SUBAPPLICATION Uebung_039b (* Spiegelabfolge V2 mit Schrittkette *)
  (* Standard: 61499-2; Description: Copyright (c) 2023 Meisterschulen am Ostbahnhof This program and the accompanying materials are made available under the terms of the Eclipse Public License 2.0 which is available at https://www.eclipse.org/legal/epl-2.0/ SPDX-License-Identifier: EPL-2.0 *)
  (* Version 1.0, 2023-10-23, Franz Höpfinger, Meisterschulen am Ostbahnhof, initial API and implementation and/or initial documentation *)
  PACKAGE Uebungen;
  IMPORT Uebungen::const::UT::DefaultPool::SoftKey_F1;
  IMPORT logiBUS::io::DQ::logiBUS_DO::Output_Q1;
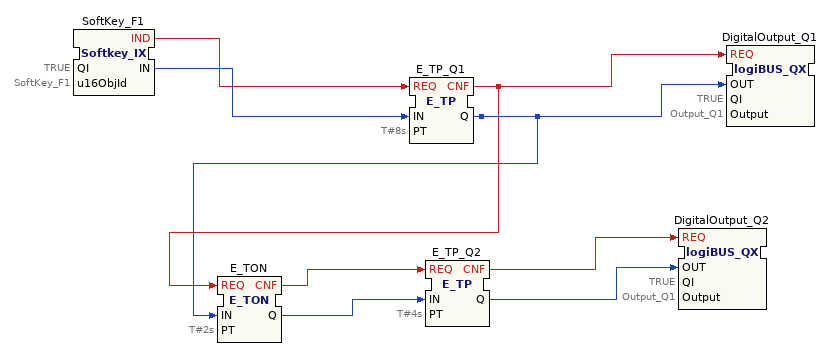
  FBS
    DigitalOutput_Q1 : logiBUS::io::DQ::logiBUS_QX(QI := TRUE, Output := Output_Q1);
    DigitalOutput_Q2 : logiBUS::io::DQ::logiBUS_QX(QI := TRUE, Output := Output_Q1);
    SoftKey_F1 : isobus::UT::io::Softkey::Softkey_IX(QI := TRUE, u16ObjId := SoftKey_F1);
    E_TP_Q1 : iec61499::events::timers::E_TP(PT := T#8s);
    E_TP_Q2 : iec61499::events::timers::E_TP(PT := T#4s);
    E_TON : iec61499::events::timers::E_TON(PT := T#2s);
  END_FBS
  EVENT_CONNECTIONS
    E_TP_Q1.CNF TO DigitalOutput_Q1.REQ;
    E_TP_Q2.CNF TO DigitalOutput_Q2.REQ;
    E_TP_Q1.CNF TO E_TON.REQ;
    E_TON.CNF TO E_TP_Q2.REQ;
    SoftKey_F1.IND TO E_TP_Q1.REQ;
  END_CONNECTIONS
  DATA_CONNECTIONS
    E_TP_Q2.Q TO DigitalOutput_Q2.OUT;
    E_TP_Q1.Q TO DigitalOutput_Q1.OUT;
    E_TP_Q1.Q TO E_TON.IN;
    E_TON.Q TO E_TP_Q2.IN;
    SoftKey_F1.IN TO E_TP_Q1.IN;
  END_CONNECTIONS
END_SUBAPPLICATION
